Universal Robots PolyScope program: Put_into_box_CB3_UR5.urp

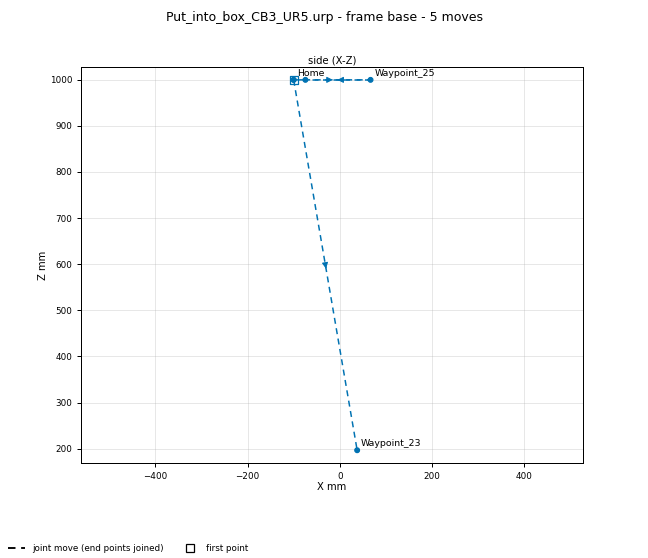
[picture p0: tool path of Put_into_box_CB3_UR5.urp in frame base, 5 of 5 moves have a stored position in this frame; points joined in program order, loops and branches not executed]
Program Put_into_box_CB3_UR5 (createdIn=1.0.0 lastSavedIn=3.2.18744 directory=/programs installation=default robotSerialNumber=2015351391)
Calibrated DH parameters: a=[0.000352, -0.161198, -0.373486, 0.00005, 0.000049, 0]; d=[0.089268, 352.477598, -320.08558, -32.281492, 0.094939, 0.082518]; alpha=[1.570728, 0.001116, -0.003686, 1.571189, -1.570572, 0]; deltaTheta=[-0.000012, 1.181849, -1.491165, 0.309495, -0.000007, 0.000025]
Robot Program (runOnlyOnce=true motionType=MoveJ speed=1.047198 acceleration=1.396263 recalculateMotions=false)
  Set NoAction (payload=0)
  MoveJ speed 10 deg/s, acceleration 80 deg/s^2 (recalculateMotions=false)
    Waypoint Home: motionParameters(blendRadius=0); TCP in base x=-99.993 y=-190.994 z=999.647 mm, rx=0.0001 ry=-2.2213 rz=2.2213 rad; joints [0, -90, 0, -90, 0, 0] deg; flange x=0.796 y=-193.992 z=1001.056 mm, rx=-0.0032 ry=2.2214 rz=-2.2182 rad
    Waypoint Waypoint_25: motionParameters(blendRadius=0); TCP in base x=66.716 y=-178.969 z=999.63 mm, rx=-0.3657 ry=2.0272 rz=-2.0272 rad; joints [20.439, -90, 0, -90, 0, 0] deg; flange x=68.491 y=-181.501 z=1001.056 mm, rx=-0.3684 ry=2.0269 rz=-2.0238 rad
    Popup Message (haltProgram=false message=Remove first bolt placed under shoulder)
    Waypoint Waypoint_26: motionParameters(blendRadius=0); TCP in base x=-74.498 y=-175.872 z=999.63 mm, rx=-0.4062 ry=-2.0012 rz=2.0011 rad; joints [-22.964, -90, 0, -90, 0, 0] deg; flange x=-74.954 y=-178.929 z=1001.056 mm, rx=-0.4042 ry=-2.0046 rz=2.0018 rad
    Popup Message (haltProgram=false message=Remove second bolt placed under shoulder                                                                      Place protective pad between arm and base joint)
    Waypoint Home: motionParameters(blendRadius=0); TCP in base x=-99.993 y=-190.994 z=999.647 mm, rx=0.0001 ry=-2.2213 rz=2.2213 rad; joints [0, -90, 0, -90, 0, 0] deg; flange x=0.796 y=-193.992 z=1001.056 mm, rx=-0.0032 ry=2.2214 rz=-2.2182 rad
    Waypoint Waypoint_23: motionParameters(blendRadius=0); TCP in base x=37.68 y=-191.036 z=196.558 mm, rx=1.2057 ry=-1.2156 rz=1.2134 rad; joints [-0.055, 3.602, -163.716, -109.496, 0.049, 0.025] deg; flange x=39.839 y=-193.023 z=195.904 mm, rx=1.2098 ry=-1.2178 rz=1.213 rad
    Popup Message (haltProgram=false message=Remove remaining bolts)
